FUNCTION_BLOCK FB_GCSpinAxisMoveVelServices EXTENDS FB_PackMLBase IMPLEMENTS I_ModuleServiceProperty
VAR_INPUT
	Ctrl : REFERENCE TO ST_GCSpinAxisMoveVelCtrl;
	Status : REFERENCE TO ST_GCSpinAxisMoveVelStatus;
	Axis_BaseUnit : REFERENCE TO FB_AxisControl;
	// The Module assigns a unique ID to this Service instance.
	ResourceOwnerId : T_ResourceOwnerId;
END_VAR

VAR_OUTPUT
END_VAR

VAR
	_StartOneShot	: R_TRIG;
	_ResetOneShot	: R_TRIG;
	_StopOneShot	: R_TRIG;
	_AbortOneShot	: R_TRIG;
	
	_ModuleMode		: T_PackMLMode;
END_VAR

// Update service state
Status.State := stOut.eStateCurrent;
Status.ActVel := Axis_BaseUnit.AxisActualVelocity;
A00_TrigCommand();

SUPER^();

ACTION A00_TrigCommand:
_StartOneShot(CLK:= Ctrl.Start);
IF _StartOneShot.Q THEN
	RequestCommand(E_PackMLCommand.Start);
END_IF

_ResetOneShot(CLK:= Ctrl.Reset);
IF _ResetOneShot.Q THEN
	RequestCommand(E_PackMLCommand.Reset);
END_IF

_StopOneShot(CLK:= Ctrl.Stop);
IF _StopOneShot.Q THEN
	RequestCommand(E_PackMLCommand.Stop);
END_IF

_AbortOneShot(CLK:= Ctrl.Abort);
IF _AbortOneShot.Q THEN
	RequestCommand(E_PackMLCommand.Abort);
END_IF
END_ACTION

METHOD PROTECTED H_OnAborted
VAR_INPUT
	bFirstScan	: BOOL;
END_VAR
// Release defensively in case an unexpected transition skipped cleanup.
Axis_BaseUnit.M_ReleaseResource(OwnerId := ResourceOwnerId);

Status.Busy := FALSE;
Status.Done := FALSE;
Status.Aborted := TRUE;

RequestCommand(E_PackMLCommand.Clear);
END_METHOD

METHOD PROTECTED H_OnAborting : E_PackMLHookResult
VAR_INPUT
	bFirstScan	: BOOL;
END_VAR

VAR
	bDone : BOOL;
	bError : BOOL;
END_VAR
H_OnAborting := E_PackMLHookResult.Busy;

// A Service that never acquired the Resource must not reset its Owner's Axis.
IF NOT Axis_BaseUnit.M_IsResourceOwner(OwnerId := ResourceOwnerId) THEN
	H_OnAborting := E_PackMLHookResult.Done;
	RETURN;
END_IF

// Withdraw MoveVelocity before resetting the Axis.
Axis_BaseUnit.M_MoveVel(
	OwnerId := ResourceOwnerId,
	Execute := FALSE,
	Ctrl.Param);
	
Axis_BaseUnit.M_Reset(
	OwnerId := ResourceOwnerId,
	Execute := TRUE,
	Done=> bDone, Error=> bError);

IF bDone THEN
	Axis_BaseUnit.M_Reset(
		OwnerId := ResourceOwnerId,
		Execute := FALSE);
	// Keep ownership until the asynchronous Reset has completed.
	Axis_BaseUnit.M_ReleaseResource(OwnerId := ResourceOwnerId);
	H_OnAborting := E_PackMLHookResult.Done;
END_IF
END_METHOD

METHOD PROTECTED H_OnClearing : E_PackMLHookResult
VAR_INPUT
	bFirstScan	: BOOL;
END_VAR

VAR
	bServoOn : BOOL;
	bError : BOOL;
	nErrorId : UDINT;
END_VAR
H_OnClearing := E_PackMLHookResult.Done;
END_METHOD

METHOD PROTECTED H_OnComplete
VAR_INPUT
	bFirstScan	: BOOL;
END_VAR
// Completing normally releases first; this is an idempotent safety net.
Axis_BaseUnit.M_ReleaseResource(OwnerId := ResourceOwnerId);

Status.Busy := FALSE;
Status.Done := TRUE;
Status.Error := FALSE;
Status.Aborted := FALSE;
Status.ErrorId := E_GCSpinAxisMoveVelErrorCode.None;

IF NOT Ctrl.Start THEN
	RequestCommand(E_PackMLCommand.Reset);
END_IF
END_METHOD

METHOD PROTECTED H_OnCompleting : E_PackMLHookResult
VAR_INPUT
	bFirstScan	: BOOL;
END_VAR
Status.Busy := FALSE;
Status.Done := TRUE;
Status.Error := FALSE;
Status.Aborted := FALSE;
Status.ErrorId := E_GCSpinAxisMoveVelErrorCode.None;

Axis_BaseUnit.M_MoveVel(
	OwnerId:= ResourceOwnerId,
	Execute:= FALSE,
	Param := Ctrl.Param);

// Release only after the active MoveVelocity request has been withdrawn.
Axis_BaseUnit.M_ReleaseResource(OwnerId := ResourceOwnerId);
H_OnCompleting := E_PackMLHookResult.Done;
END_METHOD

METHOD PROTECTED H_OnExecute : E_PackMLHookResult
VAR_INPUT
	bFirstScan	: BOOL;
END_VAR

VAR
	bDone : BOOL;
	bError : BOOL;
END_VAR
H_OnExecute := E_PackMLHookResult.Busy;

Status.Busy := TRUE;
Status.Done := FALSE;
Status.Error := FALSE;
Status.Aborted := FALSE;
Status.ErrorId := E_GCSpinAxisMoveVelErrorCode.None;

Axis_BaseUnit.M_MoveVel(
	OwnerId:= ResourceOwnerId,
	Execute:= TRUE,
	Param:= Ctrl.Param,
	InVelocity=> bDone, Error=> bError);


IF bDone THEN
	Status.Busy := FALSE;
	Status.Done := TRUE;
	H_OnExecute := E_PackMLHookResult.Done;
	RETURN;
END_IF

IF bError THEN
		Status.Error := TRUE;
		Status.ErrorId := E_GCSpinAxisMoveVelErrorCode.MoveVel_Error_During_Execute;
		
		RequestCommand(E_PackMLCommand.Stop);
END_IF
END_METHOD

METHOD PROTECTED H_OnHeld
VAR_INPUT
	bFirstScan	: BOOL;
END_VAR
// Default action hook intentionally empty. Override in derived FBs when needed.
END_METHOD

METHOD PROTECTED H_OnHolding : E_PackMLHookResult
VAR_INPUT
	bFirstScan	: BOOL;
END_VAR
// Default transient hooks complete immediately; override when work is required.
H_OnHolding := E_PackMLHookResult.Done;
END_METHOD

METHOD PROTECTED H_OnIdle
VAR_INPUT
	bFirstScan	: BOOL;
END_VAR
// Idle Services must not retain a Resource from an earlier operation.
Axis_BaseUnit.M_ReleaseResource(OwnerId := ResourceOwnerId);

Status.Busy := FALSE;
Status.Done := FALSE;
Status.Error := FALSE;
Status.Aborted := FALSE;
Status.ErrorId := E_GCSpinAxisMoveVelErrorCode.None;
END_METHOD

METHOD PROTECTED H_OnResetting : E_PackMLHookResult
VAR_INPUT
	bFirstScan	: BOOL;
END_VAR
Status.Busy := FALSE;
Status.Done := FALSE;
Status.Error := FALSE;
Status.Aborted := FALSE;
Status.ErrorId := E_GCSpinAxisMoveVelErrorCode.None;

H_OnResetting := E_PackMLHookResult.Done;
END_METHOD

METHOD PROTECTED H_OnStarting : E_PackMLHookResult
VAR_INPUT
	bFirstScan	: BOOL;
END_VAR
H_OnStarting := E_PackMLHookResult.Busy;

Status.Busy := TRUE;
Status.Done := FALSE;
Status.Error := FALSE;
Status.Aborted := FALSE;
Status.ErrorId := E_GCSpinAxisMoveVelErrorCode.None;

// Validate Service-owned data before reserving the shared BaseUnit.
IF Ctrl.Param.Velocity <= 0 THEN
	Status.Error:= TRUE;
	Status.ErrorId:= E_GCSpinAxisMoveVelErrorCode.Invalid_Param;
	RequestCommand(E_PackMLCommand.Stop);
	RETURN;
END_IF

// Resource contention is a failed Start, not a wait condition.
IF NOT Axis_BaseUnit.M_AcquireResource(OwnerId := ResourceOwnerId) THEN
	Status.Error := TRUE;
	Status.ErrorId := E_GCSpinAxisMoveVelErrorCode.Resource_Acquire_Failed_During_Starting;
	RequestCommand(E_PackMLCommand.Stop);
	RETURN;
END_IF

// Physical checks occur only after this Service owns the BaseUnit.
IF Axis_BaseUnit.AxisIsDisabled THEN
	Status.Error:= TRUE;
	Status.ErrorId:= E_GCSpinAxisMoveVelErrorCode.Axis_Not_Servo_On_During_Starting;
	RequestCommand(E_PackMLCommand.Abort);
	RETURN;
END_IF

IF Axis_BaseUnit.AxisHasJob THEN
	Status.Error:= TRUE;
	Status.ErrorId:= E_GCSpinAxisMoveVelErrorCode.Axis_Is_Busy_During_Starting;
	RequestCommand(E_PackMLCommand.Stop);
	RETURN;
END_IF

H_OnStarting := E_PackMLHookResult.Done;
END_METHOD

METHOD PROTECTED H_OnStopped
VAR_INPUT
	bFirstScan	: BOOL;
END_VAR
// Release defensively after every Stop path.
Axis_BaseUnit.M_ReleaseResource(OwnerId := ResourceOwnerId);

Status.Busy := FALSE;
Status.Done := FALSE;
Status.Aborted := TRUE;
END_METHOD

METHOD PROTECTED H_OnStopping : E_PackMLHookResult
VAR_INPUT
	bFirstScan	: BOOL;
END_VAR

VAR
	bDone : BOOL;
	bError : BOOL;
END_VAR
H_OnStopping := E_PackMLHookResult.Busy;

// Resource acquisition failures enter Stopping without owning the Axis.
IF NOT Axis_BaseUnit.M_IsResourceOwner(OwnerId := ResourceOwnerId) THEN
	H_OnStopping := E_PackMLHookResult.Done;
	RETURN;
END_IF

// Withdraw MoveVelocity before issuing the physical Stop.
Axis_BaseUnit.M_MoveVel(
	OwnerId := ResourceOwnerId,
	Execute := FALSE,
	Param:= Ctrl.Param);
	
Axis_BaseUnit.M_Stop(
	OwnerId := ResourceOwnerId,
	Execute := TRUE, 
	Deceleration:= Ctrl.Param.Deceleration,
	Done=> bDone, Error=> bError);

IF bDone THEN
	Axis_BaseUnit.M_Stop(
		OwnerId := ResourceOwnerId,
		Execute := FALSE, 
		Deceleration:= Ctrl.Param.Deceleration);
	// Ownership is released only after the asynchronous Stop has completed.
	Axis_BaseUnit.M_ReleaseResource(OwnerId := ResourceOwnerId);
	H_OnStopping := E_PackMLHookResult.Done;
	
ELSIF bError THEN
	// Throw up error
	Status.Error := TRUE;
	Status.ErrorId := E_GCSpinAxisMoveVelErrorCode.Error_While_Stop_Axis;
	
	Axis_BaseUnit.M_Stop(
		OwnerId := ResourceOwnerId,
		Execute := FALSE, 
		Deceleration:= Ctrl.Param.Deceleration);
		
	RequestCommand(E_PackMLCommand.Abort);
END_IF
END_METHOD

METHOD PROTECTED H_OnSuspended
VAR_INPUT
	bFirstScan	: BOOL;
END_VAR
// Default action hook intentionally empty. Override in derived FBs when needed.
END_METHOD

METHOD PROTECTED H_OnSuspending : E_PackMLHookResult
VAR_INPUT
	bFirstScan	: BOOL;
END_VAR
// Default transient hooks complete immediately; override when work is required.
H_OnSuspending := E_PackMLHookResult.Done;
END_METHOD

METHOD PROTECTED H_OnUndefined : E_PackMLHookResult
VAR_INPUT
	bFirstScan	: BOOL;
END_VAR
// The base FB leaves Undefined immediately unless a derived FB delays startup.
H_OnUndefined := E_PackMLHookResult.Done;
END_METHOD

METHOD PROTECTED H_OnUnholding : E_PackMLHookResult
VAR_INPUT
	bFirstScan	: BOOL;
END_VAR
// Default transient hooks complete immediately; override when work is required.
H_OnUnholding := E_PackMLHookResult.Done;
END_METHOD

METHOD PROTECTED H_OnUnsuspending : E_PackMLHookResult
VAR_INPUT
	bFirstScan	: BOOL;
END_VAR
// Default transient hooks complete immediately; override when work is required.
H_OnUnsuspending := E_PackMLHookResult.Done;
END_METHOD

PROPERTY ModuleMode : T_PackMLMode
GET
ModuleMode := _ModuleMode;
END_GET
SET
_ModuleMode := ModuleMode;
END_SET
END_PROPERTY

END_FUNCTION_BLOCK

(* stored: Version 1.1.0.1, ProductVersion 3.1.4026.18
   POU FB_GCSpinAxisMoveVelServices: Id {2d3a48e0-0a65-435f-812d-3e25cfaffe3c}, SpecialFunc None
   Folder StateAction: Id {49ed7549-95d2-4542-8c09-83ad057d2672}
   Action A00_TrigCommand: Id {9dc898aa-4aa1-4e35-9ef5-cd946bc1cd50}
   Method H_OnAborted: Id {328f5265-3f48-4442-8390-1fd00d156006}
   Method H_OnAborting: Id {8ef4724f-e418-45d4-b245-336c28b5f1de}
   Method H_OnClearing: Id {e065280f-e16e-4d87-85cf-24b54094afe6}
   Method H_OnComplete: Id {6d77d87d-d9c6-4390-a07a-5b4202d501b8}
   Method H_OnCompleting: Id {3864e1ba-9360-45a8-9d26-f1e180c8fbe5}
   Method H_OnExecute: Id {d5c34347-be90-4f5e-8be4-57798b5c5bb2}
   Method H_OnHeld: Id {290e557c-077d-4d3a-a2bb-06d511e35f5d}
   Method H_OnHolding: Id {fa63c046-0d26-4f2c-83a5-fda321bd6ee0}
   Method H_OnIdle: Id {59828899-47c9-4777-90f1-23e06ffd978a}
   Method H_OnResetting: Id {0680bc64-d1f9-407b-b6ca-83882b900618}
   Method H_OnStarting: Id {ce6c9548-1f79-4b75-96e2-343a2f8f84cb}
   Method H_OnStopped: Id {768434f7-cc85-4fdb-a507-f054649262b4}
   Method H_OnStopping: Id {b2816703-e998-4497-a19c-1d20e18f1f4c}
   Method H_OnSuspended: Id {3237239b-48f7-46dc-b2a0-07f7727d1af4}
   Method H_OnSuspending: Id {21d2483c-a2c4-4efb-8137-575165e782fc}
   Method H_OnUndefined: Id {355660e6-63b3-47e1-98ff-81122ad86689}
   Method H_OnUnholding: Id {4d791b75-be71-409c-890a-fcf31649efc0}
   Method H_OnUnsuspending: Id {cd52fade-963d-45ca-a66e-acbc7e8b9c95}
   Property ModuleMode: Id {a9425580-6a91-4e42-bb9a-1d2b8b615b56}
   Get Get: Id {0de7170a-9734-4b0e-9e84-a47c05cd839f}
   Set Set: Id {e5fffbf5-7c0f-49bc-8dd6-0eb3c9bcbadf} *)
